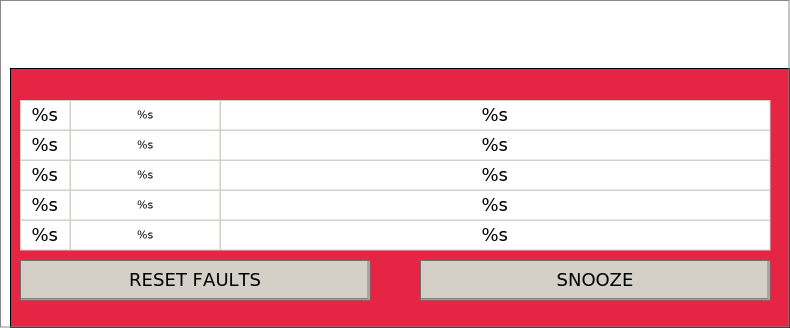
VISUALIZATION BasicMessageScreen  // 790x328
    RoundedRectangle (10,68 780x260)
    Group (20,100 754x200), invisible if: Utilities_Library.GVL_Message.bHideFaults, input disabled if: Utilities_Library.GVL_Message.bHideFaults
        Group (0,0 750x30)
            Textfield (0,0 50x30), "%s", text variable: GVL_Message.arActiveFaults[0].FaultType
            Textfield (50,0 150x30), "%s", text variable: Utilities_Library.GVL_Message.arActiveFaults[0].FullFaultId
            Textfield (200,0 550x30), "%s", text variable: Utilities_Library.GVL_Message.arActiveFaults[0].Discription
        Group (0,30 750x30)
            Textfield (0,0 50x30), "%s", text variable: Utilities_Library.GVL_Message.arActiveFaults[1].FaultType
            Textfield (50,0 150x30), "%s", text variable: Utilities_Library.GVL_Message.arActiveFaults[1].FullFaultId
            Textfield (200,0 550x30), "%s", text variable: Utilities_Library.GVL_Message.arActiveFaults[1].Discription
        Group (0,60 750x30)
            Textfield (0,0 50x30), "%s", text variable: Utilities_Library.GVL_Message.arActiveFaults[2].FaultType
            Textfield (50,0 150x30), "%s", text variable: Utilities_Library.GVL_Message.arActiveFaults[2].FullFaultId
            Textfield (200,0 550x30), "%s", text variable: Utilities_Library.GVL_Message.arActiveFaults[2].Discription
        Group (0,90 750x30)
            Textfield (0,0 50x30), "%s", text variable: Utilities_Library.GVL_Message.arActiveFaults[3].FaultType
            Textfield (50,0 150x30), "%s", text variable: Utilities_Library.GVL_Message.arActiveFaults[3].FullFaultId
            Textfield (200,0 550x30), "%s", text variable: Utilities_Library.GVL_Message.arActiveFaults[3].Discription
        Group (0,120 750x30)
            Textfield (0,0 50x30), "%s", text variable: Utilities_Library.GVL_Message.arActiveFaults[4].FaultType
            Textfield (50,0 150x30), "%s", text variable: Utilities_Library.GVL_Message.arActiveFaults[4].FullFaultId
            Textfield (200,0 550x30), "%s", text variable: Utilities_Library.GVL_Message.arActiveFaults[4].Discription
        Button (0,160 350x40), "RESET FAULTS", invisible if: Utilities_Library.GVL_Message.bHideReset, input disabled if: Utilities_Library.GVL_Message.bHideReset
            tap Utilities_Library.GVL_Message.bResetFaults
        Button (400,160 350x40), "SNOOZE"
            tap Utilities_Library.GVL_Message.bCmdSnoozeMessage
END_VISUALIZATION

(* stored: Version 1.1.0.1, ProductVersion 3.1.4024.5
   Visu BasicMessageScreen: Id {a757518a-792f-46cd-8db9-70c5517affc4} *)
